FUNCTION_BLOCK A2X_BOOL_TO_2X (* Composite FB for convert 2 BOOLS to A2X *)
  (* Standard: 61499-2; Description: Copyright (c) 2024 HR Agrartechnik GmbH This program and the accompanying materials are made available under the terms of the Eclipse Public License 2.0 which is available at https://www.eclipse.org/legal/epl-2.0/ SPDX-License-Identifier: EPL-2.0 *)
  (* Version 1.0, 2024-04-24, Franz Höpfinger, HR Agrartechnik GmbH *)
  PACKAGE adapter::conversion::unidirectional;
  IMPORT eclipse4diac::core::TypeHash;
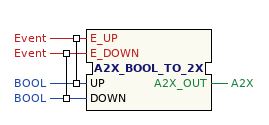
  EVENT_INPUT
    E_UP WITH UP; (* UP *)
    E_DOWN WITH DOWN; (* DOWN *)
  END_EVENT
  VAR_INPUT
    UP : BOOL; (* TRUE = forward, up, right, clockwise *)
    DOWN : BOOL; (* TRUE = backward, down, left, counter-clockwise *)
  END_VAR
  PLUGS
    A2X_OUT : adapter::types::unidirectional::A2X; (* Adapter Output *)
  END_PLUGS
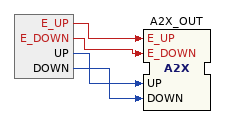
  EVENT_CONNECTIONS
    E_UP TO A2X_OUT.E_UP;
    E_DOWN TO A2X_OUT.E_DOWN;
  END_CONNECTIONS
  DATA_CONNECTIONS
    UP TO A2X_OUT.UP;
    DOWN TO A2X_OUT.DOWN;
  END_CONNECTIONS
END_FUNCTION_BLOCK
